// TIA Portal project "9_Weight_Sorting" (V19)

(* hardware
DEVICE "S7-1500/ET200MP station_1"  S7-1500 station
   slot 0: "Rail_0"  Rack  6ES7 590-1***0-0AA0
   slot 1: "PLC_1"  CPU 1513-1 PN  6ES7 513-1AL02-0AB0  V2.9
      slot 3: "CPU display_1"  6ES7591-1AA00-0AA0
      slot 32768: "PROFINET interface_1"  X1
         slot 32769: "Port_1"  X1 P1
         slot 32770: "Port_2"  X1 P2
      slot 34817: "Virtual CP interface port_1"  Virtual CP interface port  Virtual CP interface port
*)

// ===== PLC "PLC_1"  CPU 1513-1 PN =====

VAR_GLOBAL   // PLC tag table "Default tag table"
   "Network 1" AT %M0.0 : Bool;
   "Network 2" AT %M0.1 : Bool;
   "Network 3" AT %M0.3 : Bool;
   "Network 4" AT %M0.2 : Bool;
   "nw5_ase_I/P" AT %M0.4 : Bool;
   "Network 5" AT %M0.5 : Bool;
   "Network 7" AT %M1.1 : Bool;
   "Network 9" AT %M1.7 : Bool;
   "Network 5 I/P" AT %M0.6 : Bool;
   "For network 7" AT %M1.6 : Bool;
   "For network 9" AT %M2.2 : Bool;
   "Network 6 I/P(1)" AT %M1.0 : Bool;
   "Network 6" AT %M0.7 : Bool;
   "Network7_ase" AT %M1.2 : Bool;
   "Network7_are" AT %M1.5 : Bool;
   "Network8_are I/P" AT %M1.4 : Bool;
   "Network 8" AT %M1.3 : Bool;
   "Network9_ase" AT %M2.0 : Bool;
   "Network9_ale" AT %M2.1 : Bool;
   "Network10_ale" AT %M2.3 : Bool;
   "Network 10" AT %M2.4 : Bool;
END_VAR

VAR_GLOBAL   // PLC tag table "Tag table from XML_1"
   "Start" AT %I0.0 : Bool;
   "Stop" AT %I0.1 : Bool;
   "Reset" AT %I0.2 : Bool;
   "At scale" AT %I0.4 : Bool;
   "At scale exit" AT %I0.5 : Bool;
   "At forward entry" AT %I0.6 : Bool;
   "At right entry" AT %I0.7 : Bool;
   "At left entry" AT %I1.0 : Bool;
   "At exit front" AT %I1.1 : Bool;
   "At exit right" AT %I1.2 : Bool;
   "At exit left" AT %I1.3 : Bool;
   "Start light" AT %Q0.0 : Bool;
   "Stop light" AT %Q0.1 : Bool;
   "Reset Light" AT %Q0.2 : Bool;
   "Entry conveyor" AT %Q0.3 : Bool;
   "Front conveyor" AT %Q0.4 : Bool;
   "Right conveyor" AT %Q0.5 : Bool;
   "Left conveyor" AT %Q0.6 : Bool;
   "Send forward" AT %Q0.7 : Bool;
   "Send right" AT %Q1.0 : Bool;
   "Send left" AT %Q1.1 : Bool;
   "Load scale" AT %Q1.2 : Bool;
   "Weight" AT %ID30 : Real;
   "Forward count" AT %QD30 : DInt;
   "Right count" AT %QD34 : DInt;
   "Left count" AT %QD38 : DInt;
   "Weight on DP" AT %QD42 : DInt;
END_VAR

// folder: System blocks/Program resources

DATA_BLOCK "IEC_Counter_0_DB"   // DB1
{ S7_Optimized_Access := 'TRUE' }
AUTHOR : Simatic
FAMILY : IEC
NAME : CNTR
VERSION : 1.0
// stored: InstanceOfName IEC_COUNTER
"IEC_COUNTER"
BEGIN
END_DATA_BLOCK

DATA_BLOCK "IEC_Counter_0_DB_1"   // DB2
{ S7_Optimized_Access := 'TRUE' }
AUTHOR : Simatic
FAMILY : IEC
NAME : CNTR
VERSION : 1.0
// stored: InstanceOfName IEC_COUNTER
"IEC_COUNTER"
BEGIN
END_DATA_BLOCK

DATA_BLOCK "IEC_Counter_0_DB_2"   // DB3
{ S7_Optimized_Access := 'TRUE' }
AUTHOR : Simatic
FAMILY : IEC
NAME : CNTR
VERSION : 1.0
// stored: InstanceOfName IEC_COUNTER
"IEC_COUNTER"
BEGIN
END_DATA_BLOCK

// folder: (top level)

ORGANIZATION_BLOCK "Main"   // OB1, LAD, ProgramCycle
TITLE = "Main Program Sweep (Cycle)"
{ S7_Optimized_Access := 'TRUE' }
VERSION : 0.1
   VAR_INPUT
      Initial_Call : Bool;   // Initial call of this OB
      Remanence : Bool;   // =True, if remanent data are available
   END_VAR
   VAR_TEMP   // added for the SCL form of the ladder/FBD networks
      _w1 : Bool;
      _w2 : Bool;
      _w3 : Bool;
      _w4 : Bool;
   END_VAR
BEGIN

REGION Network 1: Switch ON/OFF LEDs for the start and reset button
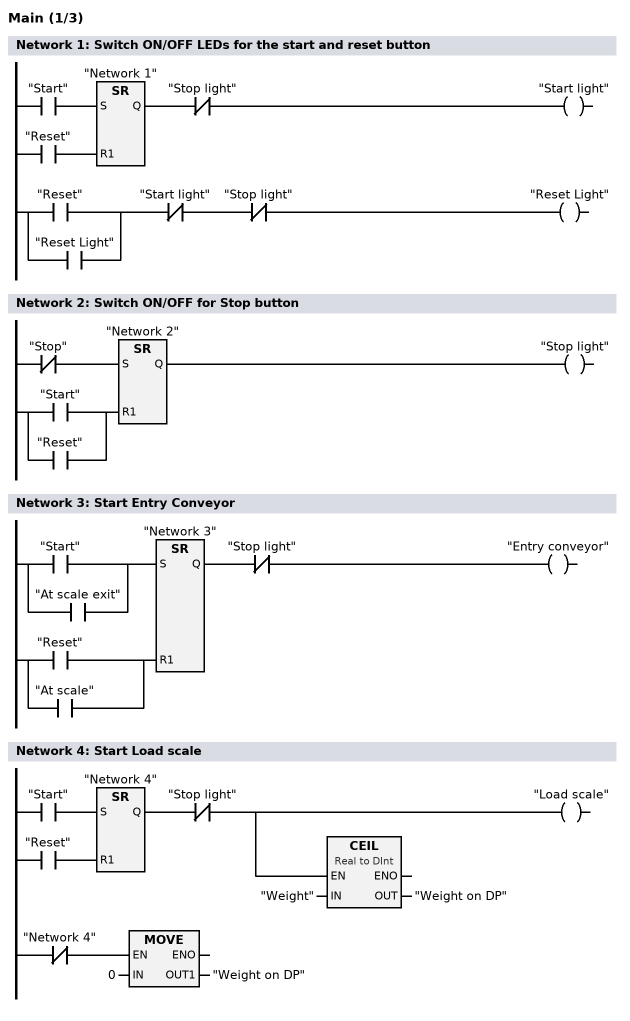
   RUNG wire#powerrail
      Contact( "Start" )
      S_SR(operand := "Network 1", r1 := wire#w1)
      I_Contact( "Stop light" )
      Coil( "Start light" )
   END_RUNG
   RUNG wire#powerrail
      Contact( "Reset" )
   END_RUNG wire#w1
   RUNG wire#powerrail
      Contact( "Reset" )
      wire#w2
      I_Contact( "Start light" )
      I_Contact( "Stop light" )
      Coil( "Reset Light" )
   END_RUNG
   RUNG wire#powerrail
      Contact( "Reset Light" )
   END_RUNG wire#w2
   // the same network as SCL:
   IF "Start" THEN
       "Network 1" := TRUE;   // SR flip-flop
   END_IF;
   IF "Reset" THEN "Network 1" := FALSE; END_IF;
   "Start light" := "Network 1" AND NOT "Stop light";
   "Reset Light" := ("Reset" OR "Reset Light") AND NOT "Start light" AND NOT "Stop light";
END_REGION

REGION Network 2: Switch ON/OFF for Stop button
   RUNG wire#powerrail
      I_Contact( "Stop" )
      S_SR(operand := "Network 2", r1 := wire#w1)
      Coil( "Stop light" )
   END_RUNG
   RUNG wire#powerrail
      Contact( "Start" )
   END_RUNG wire#w1
   RUNG wire#powerrail
      Contact( "Reset" )
   END_RUNG wire#w1
   // the same network as SCL:
   IF NOT "Stop" THEN
       "Network 2" := TRUE;   // SR flip-flop
   END_IF;
   IF "Start" OR "Reset" THEN "Network 2" := FALSE; END_IF;
   "Stop light" := "Network 2";
END_REGION

REGION Network 3: Start Entry Conveyor
   RUNG wire#powerrail
      Contact( "Start" )
      wire#w1
      S_SR(operand := "Network 3", r1 := wire#w2)
      I_Contact( "Stop light" )
      Coil( "Entry conveyor" )
   END_RUNG
   RUNG wire#powerrail
      Contact( "At scale exit" )
   END_RUNG wire#w1
   RUNG wire#powerrail
      Contact( "Reset" )
   END_RUNG wire#w2
   RUNG wire#powerrail
      Contact( "At scale" )
   END_RUNG wire#w2
   // the same network as SCL:
   IF "Start" OR "At scale exit" THEN
       "Network 3" := TRUE;   // SR flip-flop
   END_IF;
   IF "Reset" OR "At scale" THEN "Network 3" := FALSE; END_IF;
   "Entry conveyor" := "Network 3" AND NOT "Stop light";
END_REGION

REGION Network 4: Start Load scale
   IF "Start" THEN
       "Network 4" := TRUE;   // SR flip-flop
   END_IF;
   IF "Reset" THEN "Network 4" := FALSE; END_IF;
   "Load scale" := "Network 4" AND NOT "Stop light";
   IF "Load scale" THEN "Weight on DP" := CEIL("Weight"); END_IF;
   IF NOT "Network 4" THEN "Weight on DP" := 0; END_IF;
END_REGION

REGION Network 5: Start the roller
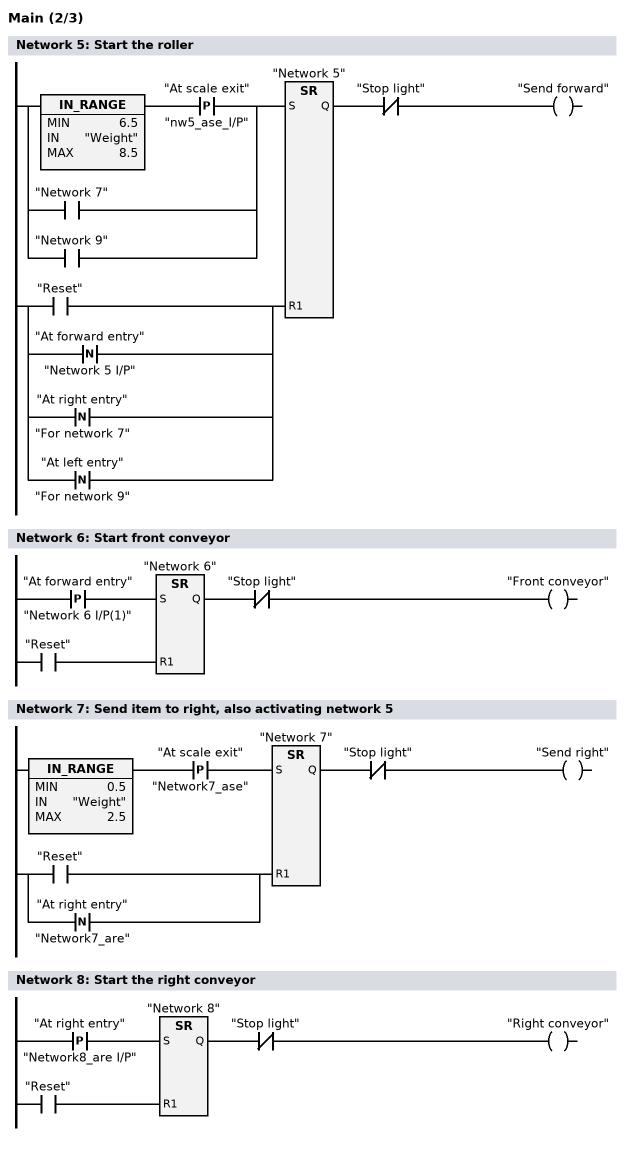
   RUNG wire#powerrail
      { S7_Templates := "SrcType := Real" } InRange(min := 6.5, in := "Weight", max := 8.5)
      P_Contact(operand := "At scale exit", bit := "nw5_ase_I/P")
      wire#w1
      S_SR(operand := "Network 5", r1 := wire#w2)
      I_Contact( "Stop light" )
      Coil( "Send forward" )
   END_RUNG
   RUNG wire#powerrail
      Contact( "Network 7" )
   END_RUNG wire#w1
   RUNG wire#powerrail
      Contact( "Network 9" )
   END_RUNG wire#w1
   RUNG wire#powerrail
      Contact( "Reset" )
   END_RUNG wire#w2
   RUNG wire#powerrail
      N_Contact(operand := "At forward entry", bit := "Network 5 I/P")
   END_RUNG wire#w2
   RUNG wire#powerrail
      N_Contact(operand := "At right entry", bit := "For network 7")
   END_RUNG wire#w2
   RUNG wire#powerrail
      N_Contact(operand := "At left entry", bit := "For network 9")
   END_RUNG wire#w2
   // the same network as SCL:
   #_w1 := (6.5 <= "Weight") AND ("Weight" <= 8.5) AND "At scale exit" AND NOT "nw5_ase_I/P";   // rising edge of "At scale exit"
   "nw5_ase_I/P" := "At scale exit";
   #_w2 := NOT "At forward entry" AND "Network 5 I/P";   // falling edge of "At forward entry"
   "Network 5 I/P" := "At forward entry";
   #_w3 := NOT "At right entry" AND "For network 7";   // falling edge of "At right entry"
   "For network 7" := "At right entry";
   #_w4 := NOT "At left entry" AND "For network 9";   // falling edge of "At left entry"
   "For network 9" := "At left entry";
   IF #_w1 OR "Network 7" OR "Network 9" THEN
       "Network 5" := TRUE;   // SR flip-flop
   END_IF;
   IF "Reset" OR #_w2 OR #_w3 OR #_w4 THEN "Network 5" := FALSE; END_IF;
   "Send forward" := "Network 5" AND NOT "Stop light";
END_REGION

REGION Network 6: Start front conveyor
   RUNG wire#powerrail
      P_Contact(operand := "At forward entry", bit := "Network 6 I/P(1)")
      S_SR(operand := "Network 6", r1 := wire#w1)
      I_Contact( "Stop light" )
      Coil( "Front conveyor" )
   END_RUNG
   RUNG wire#powerrail
      Contact( "Reset" )
   END_RUNG wire#w1
   // the same network as SCL:
   #_w1 := "At forward entry" AND NOT "Network 6 I/P(1)";   // rising edge of "At forward entry"
   "Network 6 I/P(1)" := "At forward entry";
   IF #_w1 THEN
       "Network 6" := TRUE;   // SR flip-flop
   END_IF;
   IF "Reset" THEN "Network 6" := FALSE; END_IF;
   "Front conveyor" := "Network 6" AND NOT "Stop light";
END_REGION

REGION Network 7: Send item to right, also activating network 5
   RUNG wire#powerrail
      { S7_Templates := "SrcType := Real" } InRange(min := 0.5, in := "Weight", max := 2.5)
      P_Contact(operand := "At scale exit", bit := "Network7_ase")
      S_SR(operand := "Network 7", r1 := wire#w1)
      I_Contact( "Stop light" )
      Coil( "Send right" )
   END_RUNG
   RUNG wire#powerrail
      Contact( "Reset" )
   END_RUNG wire#w1
   RUNG wire#powerrail
      N_Contact(operand := "At right entry", bit := "Network7_are")
   END_RUNG wire#w1
   // the same network as SCL:
   #_w1 := (0.5 <= "Weight") AND ("Weight" <= 2.5) AND "At scale exit" AND NOT "Network7_ase";   // rising edge of "At scale exit"
   "Network7_ase" := "At scale exit";
   #_w2 := NOT "At right entry" AND "Network7_are";   // falling edge of "At right entry"
   "Network7_are" := "At right entry";
   IF #_w1 THEN
       "Network 7" := TRUE;   // SR flip-flop
   END_IF;
   IF "Reset" OR #_w2 THEN "Network 7" := FALSE; END_IF;
   "Send right" := "Network 7" AND NOT "Stop light";
END_REGION

REGION Network 8: Start the right conveyor
   RUNG wire#powerrail
      P_Contact(operand := "At right entry", bit := "Network8_are I/P")
      S_SR(operand := "Network 8", r1 := wire#w1)
      I_Contact( "Stop light" )
      Coil( "Right conveyor" )
   END_RUNG
   RUNG wire#powerrail
      Contact( "Reset" )
   END_RUNG wire#w1
   // the same network as SCL:
   #_w1 := "At right entry" AND NOT "Network8_are I/P";   // rising edge of "At right entry"
   "Network8_are I/P" := "At right entry";
   IF #_w1 THEN
       "Network 8" := TRUE;   // SR flip-flop
   END_IF;
   IF "Reset" THEN "Network 8" := FALSE; END_IF;
   "Right conveyor" := "Network 8" AND NOT "Stop light";
END_REGION

REGION Network 9: Send item to left, also activating network 5
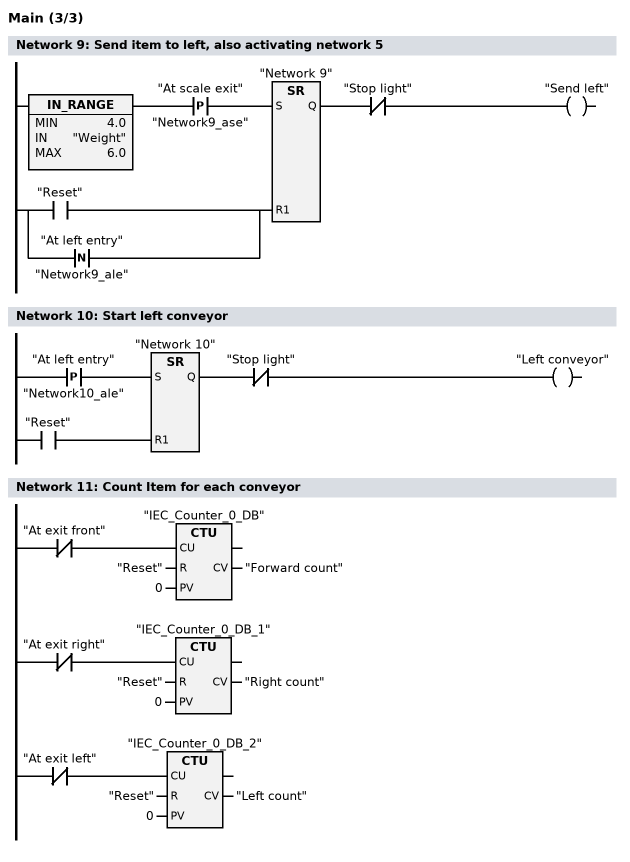
   RUNG wire#powerrail
      { S7_Templates := "SrcType := Real" } InRange(min := 4.0, in := "Weight", max := 6.0)
      P_Contact(operand := "At scale exit", bit := "Network9_ase")
      S_SR(operand := "Network 9", r1 := wire#w1)
      I_Contact( "Stop light" )
      Coil( "Send left" )
   END_RUNG
   RUNG wire#powerrail
      Contact( "Reset" )
   END_RUNG wire#w1
   RUNG wire#powerrail
      N_Contact(operand := "At left entry", bit := "Network9_ale")
   END_RUNG wire#w1
   // the same network as SCL:
   #_w1 := (4.0 <= "Weight") AND ("Weight" <= 6.0) AND "At scale exit" AND NOT "Network9_ase";   // rising edge of "At scale exit"
   "Network9_ase" := "At scale exit";
   #_w2 := NOT "At left entry" AND "Network9_ale";   // falling edge of "At left entry"
   "Network9_ale" := "At left entry";
   IF #_w1 THEN
       "Network 9" := TRUE;   // SR flip-flop
   END_IF;
   IF "Reset" OR #_w2 THEN "Network 9" := FALSE; END_IF;
   "Send left" := "Network 9" AND NOT "Stop light";
END_REGION

REGION Network 10: Start left conveyor
   RUNG wire#powerrail
      P_Contact(operand := "At left entry", bit := "Network10_ale")
      S_SR(operand := "Network 10", r1 := wire#w1)
      I_Contact( "Stop light" )
      Coil( "Left conveyor" )
   END_RUNG
   RUNG wire#powerrail
      Contact( "Reset" )
   END_RUNG wire#w1
   // the same network as SCL:
   #_w1 := "At left entry" AND NOT "Network10_ale";   // rising edge of "At left entry"
   "Network10_ale" := "At left entry";
   IF #_w1 THEN
       "Network 10" := TRUE;   // SR flip-flop
   END_IF;
   IF "Reset" THEN "Network 10" := FALSE; END_IF;
   "Left conveyor" := "Network 10" AND NOT "Stop light";
END_REGION

REGION Network 11: Count Item for each conveyor
   "IEC_Counter_0_DB".CTU(CU := NOT "At exit front", R := "Reset", PV := 0, CV => "Forward count");
   "IEC_Counter_0_DB_1".CTU(CU := NOT "At exit right", R := "Reset", PV := 0, CV => "Right count");
   "IEC_Counter_0_DB_2".CTU(CU := NOT "At exit left", R := "Reset", PV := 0, CV => "Left count");
END_REGION
END_ORGANIZATION_BLOCK